FUNCTION F_Copy : BOOL //data should of child or parent
VAR_INPUT
	Target: ANY;
	Source: ANY;
END_VAR
VAR
	nSize: UDINT;
END_VAR

IF Target.diSize > Source.diSize THEN
	nSize:= DINT_TO_UDINT(Source.diSize);
ELSE
	nSize:= DINT_TO_UDINT(Target.diSize);
END_IF

MEMCPY(
	destAddr		:= Target.pValue,
	srcAddr			:= Source.pValue,
	n				:= nSize
);

END_FUNCTION

(* stored: Version 1.1.0.1, ProductVersion 3.1.4024.12
   POU F_Copy: Id {02a7b620-6789-4498-bd8a-1f4b782ca1c5}, SpecialFunc None *)
